Fanuc KAREL source: tst_csv_read.kl

PROGRAM tst_csv_read
%NOLOCKGROUP

CONST
  CSV_NAME = 'FR:\read_data.csv'
  SAMPLE_TIME = 100

VAR
  fl : FILE
  pose : XYZWPR
  header : STRING[12]
  b : BOOLEAN

%include display.c.klt

%from display.klh %import clear, show
%from strings.klh %import pose_to_s
%include csv.klh

BEGIN
  --open csv file
  csv__read_open(CSV_NAME, fl)
  --read header
  header = csv__read_line(CSV_NAME, fl)

  --clear display
  display__clear
  --show display
  display__show
  WRITE TPDISPLAY(CR,CR)

  REPEAT
    b = csv__read_xyzwpr(CSV_NAME, fl, ',', pose)
    WRITE TPDISPLAY(pose_to_s(pose,','),CR)

    DELAY SAMPLE_TIME
  UNTIL(NOT b)

  csv__read_close(fl)

  WRITE TPDISPLAY('Read finished!',CR)

END tst_csv_read
